FUNCTION TryConvert_USINT_TO_INT : BOOL
VAR_INPUT
	in : USINT;
	out : REFERENCE TO INT;
END_VAR

out := USINT_TO_INT(in);
TryConvert_USINT_TO_INT := TRUE;

END_FUNCTION

(* stored: Version 1.1.0.1, ProductVersion 3.1.4024.12
   POU TryConvert_USINT_TO_INT: Id {14bd9e63-5212-488f-95f8-e5d655bec00a}, SpecialFunc None *)
